FUNCTION_BLOCK ABSTRACT Communicator EXTENDS TC.ToolkitObject
VAR_INPUT
	CycleInterval : TIME; 
	CyclicMode : BOOL; 
END_VAR
VAR_OUTPUT
	{attribute 'OPC.UA.DA.Access' := '1'}	
	Configured : BOOL;
	{attribute 'OPC.UA.DA.Access' := '1'}	
	CycleCount : ULINT;
	{attribute 'OPC.UA.DA.Access' := '1'}	
	DefaultOperationTimeout : TIME; 
END_VAR
VAR
	{attribute 'OPC.UA.DA' := '0'}	
	_InitialCyclicMode : BOOL; 
	{attribute 'OPC.UA.DA' := '0'}	
	_LastException : Exception;
END_VAR

{attribute 'monitoring' := 'call'}
{attribute 'OPC.UA.DA' := '1'}
{attribute 'OPC.UA.DA.Property' := '1'}
PROPERTY ABSTRACT Busy : BOOL
GET
END_GET
END_PROPERTY

METHOD Clear : BOOL
VAR_OUTPUT
	exception : Exception;
END_VAR
IF Busy THEN
	ExceptionHelper.Throw(0, "Communicator is busy", __POUNAME(), ClassName, CurrentNamespace.Name, __POSITION());
	RETURN;
END_IF

AdsLogger.LogMessage(LOGGING_LEVEL.INFORMATION, "---Communicator.Clear");

CycleCount := 0;
_LastException.Clear();

Clear := InternalClear(exception => exception);
END_METHOD

PROPERTY ABSTRACT CommunicationTypeName : STRING
GET
END_GET
END_PROPERTY

METHOD FINAL Configure : BOOL
VAR_INPUT
	settings : REFERENCE TO CommunicationSettings;
END_VAR
VAR_OUTPUT
	exception : Exception;
END_VAR
IF Busy THEN
	ExceptionHelper.Throw(0, "Communicator is busy", __POUNAME(), ClassName, CurrentNamespace.Name, __POSITION());
	RETURN;
END_IF

IF NOT __ISVALIDREF(settings) THEN
	ExceptionHelper.Throw(0, "Parameter 'settings' has not been specified", __POUNAME(), ClassName, CurrentNamespace.Name, __POSITION());
	RETURN;
END_IF

IF CommunicationTypeName <> settings.CommunicationTypeName THEN
	ExceptionHelper.Throw(0, WStringHelper.Concat4("Communicator and communication settings are incompatible because has different CommunicationTypeName: ", TO_WSTRING(CommunicationTypeName), " and ", TO_WSTRING(settings.CommunicationTypeName)), __POUNAME(), ClassName, CurrentNamespace.Name, __POSITION());
	RETURN;
END_IF

IF settings.DefaultOperationTimeout > T#0S THEN
	DefaultOperationTimeout := settings.DefaultOperationTimeout;
ELSE	
	DefaultOperationTimeout := Tc2_System.DEFAULT_ADS_TIMEOUT;
END_IF

AdsLogger.LogMessage(LOGGING_LEVEL.INFORMATION, "---Communicator.Configure");

Configured := Configure := InternalConfigure(settings, exception => exception);
END_METHOD

{attribute 'monitoring' := 'call'}
{attribute 'OPC.UA.DA' := '1'}
{attribute 'OPC.UA.DA.Property' := '1'}
PROPERTY DataProcessed : BOOL
GET
END_GET
END_PROPERTY

{attribute 'monitoring' := 'call'}
{attribute 'OPC.UA.DA' := '1'}
{attribute 'OPC.UA.DA.Property' := '1'}
PROPERTY Error : BOOL
GET
END_GET
END_PROPERTY

METHOD ABSTRACT Execute
END_METHOD

METHOD PROTECTED GetOperationTimeout : TIME
VAR_INPUT
	operationTimeout : TIME;
END_VAR
IF operationTimeout = T#0S THEN
	getOperationTimeout := DefaultOperationTimeout;
ELSE
	getOperationTimeout := operationTimeout;
END_IF
END_METHOD

METHOD PROTECTED ABSTRACT InternalClear : BOOL
VAR_OUTPUT
	exception : Exception;
END_VAR
END_METHOD

METHOD PROTECTED ABSTRACT InternalConfigure : BOOL
VAR_INPUT
	settings : REFERENCE TO CommunicationSettings;
END_VAR
VAR_OUTPUT
	exception : Exception;
END_VAR
END_METHOD

METHOD PROTECTED ABSTRACT InternalStart : BOOL
VAR_OUTPUT
	exception : Exception;
END_VAR
END_METHOD

METHOD PROTECTED ABSTRACT InternalStop
END_METHOD

{attribute 'monitoring' := 'call'}
{attribute 'OPC.UA.DA.Property' := '1'}
{attribute 'OPC.UA.DA.Access' := '1'}
PROPERTY FINAL LastException : REFERENCE TO Exception
GET
LastException REF= _LastException;
END_GET
END_PROPERTY

METHOD FINAL Start : BOOL
VAR_OUTPUT
	exception : Exception;
END_VAR
IF Busy THEN
	ExceptionHelper.Throw(0, "Communicator is busy", __POUNAME(), ClassName, CurrentNamespace.Name, __POSITION());
	RETURN;
END_IF

AdsLogger.LogMessage(LOGGING_LEVEL.INFORMATION, "---Communicator.Start");

CycleCount := 0;
_LastException.Clear();

Start := InternalStart(exception => exception);
END_METHOD

METHOD FINAL Stop
IF Busy THEN
	AdsLogger.LogMessage(LOGGING_LEVEL.INFORMATION, "---Communicator.Stop");
		
	InternalStop();
END_IF
END_METHOD

PROPERTY ABSTRACT VariablesCount : DINT
GET
END_GET
END_PROPERTY

END_FUNCTION_BLOCK

(* stored: Version 1.1.0.1
   POU Communicator: Id {c51ea328-1ad2-4150-bf21-69a5a6298ef3}, SpecialFunc None
   Folder Internal methods to override: Id {433e7843-11fb-015f-3b11-10f8d73326b0}
   Folder Service methods: Id {28df0cb1-f445-0eae-3e86-2f4f177a0128}
   Property Busy: Id {acbc8522-7f92-46a6-9a7a-4c37eb222979}
   Get Get: Id {6f3f9f49-e8b5-4432-b9e5-c73b5df26ea4}
   Method Clear: Id {dfc1da11-3da6-4078-befc-749dc8cc9443}
   Property CommunicationTypeName: Id {c74b7738-018d-42f7-93b9-781d86a80ce8}
   Get Get: Id {029cc94a-5457-4247-9fed-6bae629f55aa}
   Method Configure: Id {d92b918b-a981-42f5-aa1c-968b19d6d620}
   Property DataProcessed: Id {ec69b158-0bc9-4b4e-8455-43d8b34fba09}
   Get Get: Id {88b9b370-37b2-4a92-ae5b-718815693bd3}
   Property Error: Id {ddd9647a-1280-4bcd-ae2d-43cd5ba67f11}
   Get Get: Id {63a76cc6-6148-4884-bdc9-eb791c637011}
   Method Execute: Id {4e0fec5f-09f0-44f7-b315-fd6fd7524589}
   Method GetOperationTimeout: Id {98d48482-808e-0512-031b-25a7b489ed20}
   Method InternalClear: Id {1d6f5521-f2f3-448a-bdae-b01ea63a7bc1}
   Method InternalConfigure: Id {963a6689-24ee-4add-a784-7f449c9755ce}
   Method InternalStart: Id {771ca01c-edd8-4b11-82bb-00fb10add390}
   Method InternalStop: Id {5e07a7af-614c-4e84-8c8c-d0cc26f2ef34}
   Property LastException: Id {4bfb2624-14b2-4b1e-aae8-90c27a1dfa77}
   Get Get: Id {5c679964-232b-4b80-8391-742c5df38c63}
   Method Start: Id {082abe1b-0d7b-4cbf-98fe-ee5338ebfb32}
   Method Stop: Id {bede61f5-c962-4f45-a6e8-adbfdd89db64}
   Property VariablesCount: Id {55e54645-3cc7-0e9c-0086-64bb68ad623e}
   Get Get: Id {c8db8f1b-519d-0c52-2baf-549346b30aee} *)
